// TIA Portal V18 export
TYPE "LGasp_type_quote_impilaggio"
// stored: IsFailsafeCompliant false
   STRUCT
      index_riga : DInt;   // indice di riga [1..riga max]
      index_colonna : DInt;   // indice di colonna [1..colonna max]
      X : LReal;   // [mm] quota in X pezzo
      Y : LReal;   // [mm] quota in Y pezzo
      Z : LReal;   // [mm] quota in Z pezzo
   END_STRUCT;
END_TYPE
